(* Logix 5000 project; controller Reto3_PID Emulate 5570 rev 30.12; software revision 30.00 *)

TASK Alarma (periodic, rate 10 ms, priority 10, watchdog 500 ms) : Alarma_sensores
TASK Escalizaciones (periodic, rate 10 ms, priority 10, watchdog 500 ms) : Escalizacion_sensores
TASK MainTask (continuous, watchdog 500 ms) : MainProgram

MODULES
   Local : Emulate 5570 (ICP 2, rev 30.12)
END_MODULES

VAR_GLOBAL   (* controller tags *)
   A0_0 : REAL;
   AO_1 : REAL;
   Bandera_Flujo : BOOL;
   Bandera_Nivel : BOOL;
   Control_Flujo : PID;
   Control_Nivel : PID := (CTL := 1053312, NOZC := 1, OLH := 1, DVPA := 1, PVHA := 1, KP := 1.0, KI := 1.0, KD := 0.5, MAXS := 300.0, SO := 100.0, MAXO := 100.0, UPD := 0.01, ERR := 11.629463, MAXI := 10.0, MAXCV := 300.0, MAXTIE := 100.0, DATA[0] := 95.998795, DATA[1] := -430.4896, DATA[2] := 80.7168, DATA[3] := 11.629463, DATA[4] := 92.34626, DATA[5] := 0.33333334, DATA[6] := 30.0, DATA[7] := 2.1, DATA[8] := 1.0, DATA[9] := 1.0, DATA[10] := 0.5, DATA[11] := 1.0, DATA[12] := 1.0, DATA[13] := 0.5, DATA[15] := 3.0, DATA[16] := 1.0);
   CT_SelectFlujo : BOOL;
   CT_SelectNivel : BOOL := 1;
   CT_SetPoint : REAL;
   CT_T_Flujo : REAL;
   CT_T_Nivel : REAL := 0.38047975;
   CT_VDescarga : REAL := 300.0;
   CT_Vllenado : REAL := 5.0;
   Flujo_tanque : REAL;
   INT_OUT_0 : DINT;
   INT_OUT_1 : DINT;
   Mult_SetPoint : REAL;
   Mult_Tflujo : REAL;
   Mult_Tnivel : REAL := 114.14393;
   Nivel_H : BOOL;
   Nivel_HH : BOOL;
   Nivel_tanque : REAL := 11.414392;
   Set_point : REAL;
   Set_point_Flujo : REAL;
   Set_point_Nivel : REAL;
   Start : BOOL;
   Stop : BOOL := 1;
END_VAR

PROGRAM Alarma_sensores   (* main routine Alarma_rutina *)

ROUTINE Alarma_rutina   (* ladder *)
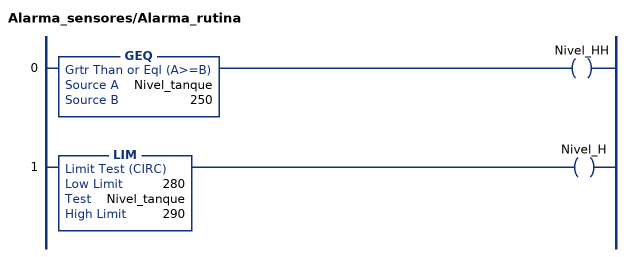
   0: GEQ(Nivel_tanque,250)OTE(Nivel_HH);
   1: LIM(280,Nivel_tanque,290)OTE(Nivel_H);
END_ROUTINE
END_PROGRAM

PROGRAM Escalizacion_sensores   (* main routine Escalizacion_rutina *)

ROUTINE Escalizacion_rutina   (* ladder *)
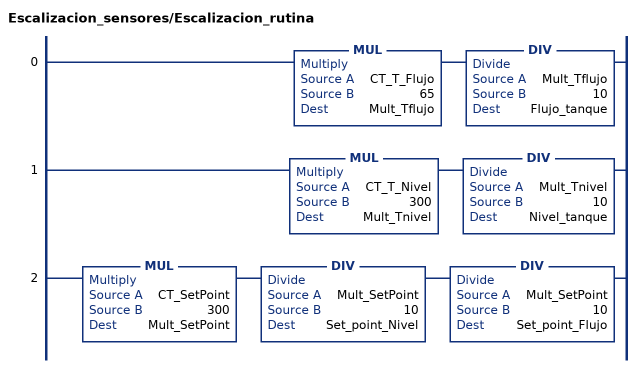
   0: MUL(CT_T_Flujo,65,Mult_Tflujo)DIV(Mult_Tflujo,10,Flujo_tanque);
   1: MUL(CT_T_Nivel,300,Mult_Tnivel)DIV(Mult_Tnivel,10,Nivel_tanque);
   2: MUL(CT_SetPoint,300,Mult_SetPoint)DIV(Mult_SetPoint,10,Set_point_Nivel)DIV(Mult_SetPoint,10,Set_point_Flujo);
END_ROUTINE
END_PROGRAM

PROGRAM MainProgram   (* main routine MainRoutine *)

ROUTINE Flujo   (* ladder *)
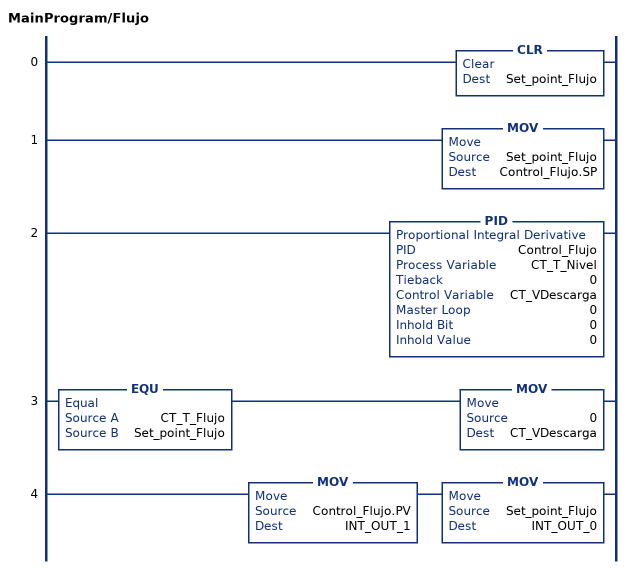
   0: CLR(Set_point_Flujo);
   1: MOV(Set_point_Flujo,Control_Flujo.SP);
   2: PID(Control_Flujo,CT_T_Nivel,0,CT_VDescarga,0,0,0);
   3: EQU(CT_T_Flujo,Set_point_Flujo)MOV(0,CT_VDescarga);
   4: MOV(Control_Flujo.PV,INT_OUT_1)MOV(Set_point_Flujo,INT_OUT_0);
END_ROUTINE

ROUTINE MainRoutine   (* ladder *)
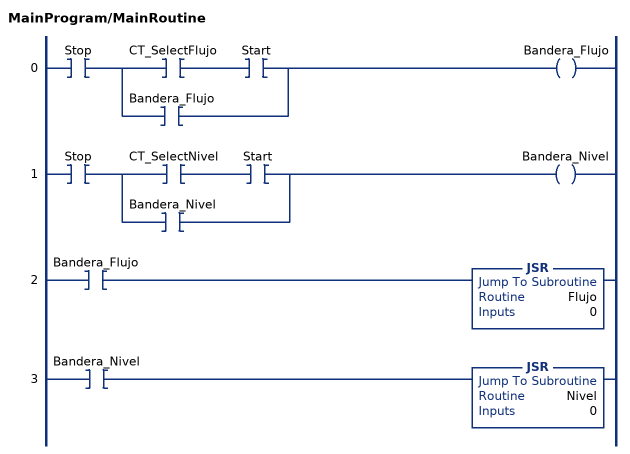
   0: XIC(Stop)[XIC(CT_SelectFlujo) XIC(Start) ,XIC(Bandera_Flujo) ]OTE(Bandera_Flujo);
   1: XIC(Stop)[XIC(CT_SelectNivel) XIC(Start) ,XIC(Bandera_Nivel) ]OTE(Bandera_Nivel);
   2: XIC(Bandera_Flujo)JSR(Flujo,0);
   3: XIC(Bandera_Nivel)JSR(Nivel,0);
END_ROUTINE

ROUTINE Nivel   (* ladder *)
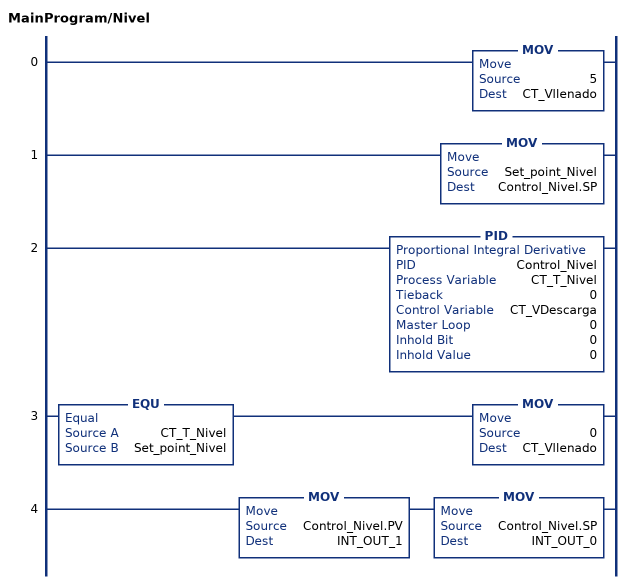
   0: MOV(5,CT_Vllenado);
   1: MOV(Set_point_Nivel,Control_Nivel.SP);
   2: PID(Control_Nivel,CT_T_Nivel,0,CT_VDescarga,0,0,0);
   3: EQU(CT_T_Nivel,Set_point_Nivel)MOV(0,CT_Vllenado);
   4: MOV(Control_Nivel.PV,INT_OUT_1)MOV(Control_Nivel.SP,INT_OUT_0);
END_ROUTINE
END_PROGRAM
